FUNCTION Buffer_Layout_Set_USInt_Array : UINT
VAR_INPUT
END_VAR
VAR
END_VAR

END_FUNCTION

(* stored: Version 1.1.0.1, ProductVersion 3.1.4024.10
   POU Buffer_Layout_Set_USInt_Array: Id {37bfa2a9-e120-4901-b10b-08a05e13ad83}, SpecialFunc None *)
